(* IEC 61131-3 sources: FactoryIO-PLC/examples/testbed, 4 files *)

(* ---- FT_con01.st ---- *)
PROGRAM Cell1
  VAR
    R1_front AT %IX0.2 : BOOL := true;
    R1_rear AT %IX0.3 : BOOL := true;
    C1_endIR AT %IX0.4 : BOOL := true;
    C1_startIR AT %IX0.5 : BOOL := true;
    Main AT %IX0.6 : BOOL := false;
    R1_fwd_motor AT %QX0.2 : BOOL := true;
    R1_bwd_motor AT %QX0.3 : BOOL := true;
    C1_motor AT %QX0.4 : BOOL := true;
  END_VAR
  VAR
    C1_working : BOOL := false;
  END_VAR
  VAR
    C1_working_int AT %MD1 : DINT := 0;
  END_VAR
  VAR
    R1_in_transit : BOOL := false;
  END_VAR
  VAR
    R1_in_transit_int AT %MD3 : DINT := 0;
  END_VAR
  VAR
    R1_fwd : BOOL := false;
  END_VAR
  VAR
    R1_fwd_int AT %MD4 : DINT := 0;
  END_VAR
  VAR
    R1_bwd : BOOL := false;
  END_VAR
  VAR
    R1_bwd_int AT %MD5 : DINT := 0;
  END_VAR
  VAR
    Timer_in_transit : TON;
    BOOL_TO_DINT27_ENO : BOOL;
    BOOL_TO_DINT27_OUT : DINT;
    BOOL_TO_DINT37_ENO : BOOL;
    BOOL_TO_DINT37_OUT : DINT;
    BOOL_TO_DINT61_ENO : BOOL;
    BOOL_TO_DINT61_OUT : DINT;
    BOOL_TO_DINT67_ENO : BOOL;
    BOOL_TO_DINT67_OUT : DINT;
  END_VAR

  IF NOT(C1_startIR) THEN
    C1_working := TRUE; (*set*)
  END_IF;
  C1_motor := NOT(C1_working AND NOT(Main));
  IF NOT(C1_endIR) THEN
    R1_in_transit := TRUE; (*set*)
  END_IF;
  Timer_in_transit(IN := R1_in_transit AND C1_working, PT := T#1000ms);
  IF Timer_in_transit.Q THEN
    R1_fwd := TRUE; (*set*)
  END_IF;
  IF Timer_in_transit.Q THEN
    C1_working := FALSE; (*reset*)
  END_IF;
  IF Timer_in_transit.Q THEN
    R1_in_transit := FALSE; (*reset*)
  END_IF;
  R1_fwd_motor := NOT(R1_fwd AND NOT(Main));
  IF NOT(R1_front) AND R1_fwd THEN
    R1_bwd := TRUE; (*set*)
  END_IF;
  IF NOT(R1_front) AND R1_fwd THEN
    R1_fwd := FALSE; (*reset*)
  END_IF;
  R1_bwd_motor := NOT(R1_bwd AND NOT(Main));
  IF NOT(R1_rear) AND R1_bwd THEN
    R1_bwd := FALSE; (*reset*)
  END_IF;
  BOOL_TO_DINT27_OUT := BOOL_TO_DINT(EN := TRUE, IN := C1_working, ENO => BOOL_TO_DINT27_ENO);
  C1_working_int := BOOL_TO_DINT27_OUT;
  BOOL_TO_DINT37_OUT := BOOL_TO_DINT(EN := TRUE, IN := R1_in_transit, ENO => BOOL_TO_DINT37_ENO);
  R1_in_transit_int := BOOL_TO_DINT37_OUT;
  BOOL_TO_DINT61_OUT := BOOL_TO_DINT(EN := TRUE, IN := R1_fwd, ENO => BOOL_TO_DINT61_ENO);
  R1_fwd_int := BOOL_TO_DINT61_OUT;
  BOOL_TO_DINT67_OUT := BOOL_TO_DINT(EN := TRUE, IN := R1_bwd, ENO => BOOL_TO_DINT67_ENO);
  R1_bwd_int := BOOL_TO_DINT67_OUT;
END_PROGRAM

CONFIGURATION Config0

  RESOURCE Res0 ON PLC
    TASK TaskMain(INTERVAL := T#50ms,PRIORITY := 0);
    PROGRAM Inst0 WITH TaskMain : Cell1;
  END_RESOURCE
END_CONFIGURATION

(* ---- FT_con02.st ---- *)
PROGRAM Cell2
  VAR
    C1_IR AT %IX0.3 : BOOL := true;
    M1_IR AT %IX0.4 : BOOL := true;
    Main AT %IX0.6 : BOOL := true;
    M1_motor AT %QX0.2 : BOOL := true;
    C2_motor AT %QX0.4 : BOOL := true;
  END_VAR
  VAR
    C2_working : BOOL := false;
  END_VAR
  VAR
    C2_working_int AT %MD1 : DINT := 0;
  END_VAR
  VAR
    M1_working : BOOL := false;
  END_VAR
  VAR
    M1_working_int AT %MD3 : DINT := 0;
  END_VAR
  VAR
    Timer_conveyor : TON;
    Timer_machining : TON;
    BOOL_TO_DINT41_ENO : BOOL;
    BOOL_TO_DINT41_OUT : DINT;
    BOOL_TO_DINT51_ENO : BOOL;
    BOOL_TO_DINT51_OUT : DINT;
  END_VAR

  IF NOT(C1_IR) THEN
    C2_working := TRUE; (*set*)
  END_IF;
  C2_motor := NOT(C2_working AND NOT(Main));
  IF NOT(M1_IR) AND C2_working THEN
    M1_working := TRUE; (*set*)
  END_IF;
  IF NOT(M1_IR) AND C2_working THEN
    C2_working := FALSE; (*reset*)
  END_IF;
  M1_motor := NOT(M1_working AND NOT(Main));
  Timer_machining(IN := M1_working, PT := T#3000ms);
  IF Timer_machining.Q THEN
    C2_working := TRUE; (*set*)
  END_IF;
  IF Timer_machining.Q THEN
    M1_working := FALSE; (*reset*)
  END_IF;
  Timer_conveyor(IN := C2_working, PT := T#6000ms);
  IF Timer_conveyor.Q THEN
    C2_working := FALSE; (*reset*)
  END_IF;
  BOOL_TO_DINT41_OUT := BOOL_TO_DINT(EN := TRUE, IN := C2_working, ENO => BOOL_TO_DINT41_ENO);
  C2_working_int := BOOL_TO_DINT41_OUT;
  BOOL_TO_DINT51_OUT := BOOL_TO_DINT(EN := TRUE, IN := M1_working, ENO => BOOL_TO_DINT51_ENO);
  M1_working_int := BOOL_TO_DINT51_OUT;
END_PROGRAM

CONFIGURATION Config0

  RESOURCE Res0 ON PLC
    TASK TaskMain(INTERVAL := T#50ms,PRIORITY := 0);
    PROGRAM Inst0 WITH TaskMain : Cell2;
  END_RESOURCE
END_CONFIGURATION

(* ---- FT_con03.st ---- *)
PROGRAM Cell3
  VAR
    C2_IR AT %IX0.3 : BOOL := true;
    M2_IR AT %IX0.4 : BOOL := true;
    Main AT %IX0.6 : BOOL := true;
    M2_motor AT %QX0.2 : BOOL := true;
    C3_motor AT %QX0.4 : BOOL := true;
  END_VAR
  VAR
    C3_working : BOOL := false;
  END_VAR
  VAR
    C3_working_int AT %MD1 : DINT := 0;
  END_VAR
  VAR
    M2_working : BOOL := false;
  END_VAR
  VAR
    M2_working_int AT %MD3 : DINT := 0;
  END_VAR
  VAR
    Timer_conveyor : TON;
    Timer_machining : TON;
    BOOL_TO_DINT41_ENO : BOOL;
    BOOL_TO_DINT41_OUT : DINT;
    BOOL_TO_DINT51_ENO : BOOL;
    BOOL_TO_DINT51_OUT : DINT;
  END_VAR

  IF NOT(C2_IR) THEN
    C3_working := TRUE; (*set*)
  END_IF;
  C3_motor := NOT(C3_working AND NOT(Main));
  IF NOT(M2_IR) AND C3_working THEN
    M2_working := TRUE; (*set*)
  END_IF;
  IF NOT(M2_IR) AND C3_working THEN
    C3_working := FALSE; (*reset*)
  END_IF;
  M2_motor := NOT(M2_working AND NOT(Main));
  Timer_machining(IN := M2_working, PT := T#3000ms);
  IF Timer_machining.Q THEN
    C3_working := TRUE; (*set*)
  END_IF;
  IF Timer_machining.Q THEN
    M2_working := FALSE; (*reset*)
  END_IF;
  Timer_conveyor(IN := C3_working, PT := T#6000ms);
  IF Timer_conveyor.Q THEN
    C3_working := FALSE; (*reset*)
  END_IF;
  BOOL_TO_DINT41_OUT := BOOL_TO_DINT(EN := TRUE, IN := C3_working, ENO => BOOL_TO_DINT41_ENO);
  C3_working_int := BOOL_TO_DINT41_OUT;
  BOOL_TO_DINT51_OUT := BOOL_TO_DINT(EN := TRUE, IN := M2_working, ENO => BOOL_TO_DINT51_ENO);
  M2_working_int := BOOL_TO_DINT51_OUT;
END_PROGRAM

CONFIGURATION Config0

  RESOURCE Res0 ON PLC
    TASK TaskMain(INTERVAL := T#50ms,PRIORITY := 0);
    PROGRAM Inst0 WITH TaskMain : Cell3;
  END_RESOURCE
END_CONFIGURATION

(* ---- FT_con04.st ---- *)
PROGRAM Cell4
  VAR
    R2_front AT %IX0.2 : BOOL := true;
    R2_rear AT %IX0.3 : BOOL := true;
    C4_endIR AT %IX0.4 : BOOL := true;
    C3_IR AT %IX0.5 : BOOL := true;
    Main AT %IX0.6 : BOOL := false;
    R2_fwd_motor AT %QX0.2 : BOOL := true;
    R2_bwd_motor AT %QX0.3 : BOOL := true;
    C4_motor AT %QX0.4 : BOOL := true;
  END_VAR
  VAR
    C4_working : BOOL := false;
  END_VAR
  VAR
    C4_working_int AT %MD1 : DINT := 0;
  END_VAR
  VAR
    R2_in_transit : BOOL := false;
  END_VAR
  VAR
    R2_in_transit_int AT %MD3 : DINT := 0;
  END_VAR
  VAR
    R2_fwd : BOOL := false;
  END_VAR
  VAR
    R2_fwd_int AT %MD4 : DINT := 0;
  END_VAR
  VAR
    R2_bwd : BOOL := false;
  END_VAR
  VAR
    R2_bwd_int AT %MD5 : DINT := 0;
  END_VAR
  VAR
    Timer_in_transit : TON;
    BOOL_TO_DINT49_ENO : BOOL;
    BOOL_TO_DINT49_OUT : DINT;
    BOOL_TO_DINT64_ENO : BOOL;
    BOOL_TO_DINT64_OUT : DINT;
    BOOL_TO_DINT61_ENO : BOOL;
    BOOL_TO_DINT61_OUT : DINT;
    BOOL_TO_DINT67_ENO : BOOL;
    BOOL_TO_DINT67_OUT : DINT;
  END_VAR

  IF NOT(C3_IR) THEN
    R2_in_transit := TRUE; (*set*)
  END_IF;
  Timer_in_transit(IN := R2_in_transit, PT := T#4500ms);
  IF Timer_in_transit.Q THEN
    R2_fwd := TRUE; (*set*)
  END_IF;
  IF Timer_in_transit.Q THEN
    C4_working := TRUE; (*set*)
  END_IF;
  IF Timer_in_transit.Q THEN
    R2_in_transit := FALSE; (*reset*)
  END_IF;
  R2_fwd_motor := NOT(R2_fwd AND NOT(Main));
  IF NOT(R2_front) AND R2_fwd THEN
    R2_bwd := TRUE; (*set*)
  END_IF;
  IF NOT(R2_front) AND R2_fwd THEN
    R2_fwd := FALSE; (*reset*)
  END_IF;
  R2_bwd_motor := NOT(R2_bwd AND NOT(Main) AND TRUE);
  IF NOT(R2_rear) AND R2_bwd THEN
    R2_bwd := FALSE; (*reset*)
  END_IF;
  C4_motor := NOT(C4_working AND NOT(Main));
  IF NOT(C4_endIR) AND C4_working THEN
    C4_working := FALSE; (*reset*)
  END_IF;
  BOOL_TO_DINT49_OUT := BOOL_TO_DINT(EN := TRUE, IN := C4_working, ENO => BOOL_TO_DINT49_ENO);
  C4_working_int := BOOL_TO_DINT49_OUT;
  BOOL_TO_DINT64_OUT := BOOL_TO_DINT(EN := TRUE, IN := R2_in_transit, ENO => BOOL_TO_DINT64_ENO);
  R2_in_transit_int := BOOL_TO_DINT64_OUT;
  BOOL_TO_DINT61_OUT := BOOL_TO_DINT(EN := TRUE, IN := R2_fwd, ENO => BOOL_TO_DINT61_ENO);
  R2_fwd_int := BOOL_TO_DINT61_OUT;
  BOOL_TO_DINT67_OUT := BOOL_TO_DINT(EN := TRUE, IN := R2_bwd, ENO => BOOL_TO_DINT67_ENO);
  R2_bwd_int := BOOL_TO_DINT67_OUT;
END_PROGRAM

CONFIGURATION Config0

  RESOURCE Res0 ON PLC
    TASK TaskMain(INTERVAL := T#50ms,PRIORITY := 0);
    PROGRAM Inst0 WITH TaskMain : Cell4;
  END_RESOURCE
END_CONFIGURATION
